FUNCTION_BLOCK Room_State_Disabled EXTENDS Room_State
VAR_INPUT
END_VAR
VAR_OUTPUT
END_VAR
VAR
END_VAR

METHOD OnExecute
IF NOT _ctx.hmi.bDisable THEN
	_ctx.state.iMgr.Request(_ctx.state.iIdle);
END_IF
END_METHOD

METHOD OnEntry
_ctx.io.bOpenValves := TRUE;

_ctx.priv.bActive := FALSE;
_ctx.priv.bReady := FALSE;

_ctx.hmi.sStatusText := 'ROOM DISABLED!';
_ctx.hmi.nStatusColor := COL.RED.Raw;

_ctx.hmi.bHideReset := TRUE;
END_METHOD

END_FUNCTION_BLOCK

(* stored: Version 1.1.0.1
   POU Room_State_Disabled: Id {233cb2a4-a188-4d83-a20b-e18c2158eca6}, SpecialFunc None
   Method OnExecute: Id {77eb3e2f-d766-45f5-844e-dd3b61e6835e}
   Method OnInit: Id {f389e261-ef83-454d-a100-de95232fb4c4} *)
